FUNCTION_BLOCK FB_Example2

VAR
	fbRead1     :  FB_ReadAdsSymByName;
	bEnable     : BOOL;
	sSymbol     : STRING := 'GVL_Config.arrRack[1]';
	stStorageSlot : ST_StorageSlot;
	eComMode    :  E_AdsComMode := eAdsComModeFastCom;
	bBusy       : BOOL;
    bError      : BOOL;
    nErrId      : UDINT;
	bExecute: BOOL;
	fbTimer : TON := (PT := T#100MS); // Adjust the speed here
END_VAR


fbTimer(IN := NOT fbTimer.Q); // This creates a self-resetting pulse

IF fbTimer.Q THEN
    bEnable := TRUE; // Trigger your FB_ReadAdsSymByName
END_IF

	fbRead1(
	bRead:= bEnable, 
	sNetId:= '', 
	nPort:= 852, 
	sVarName:= sSymbol, 
	nDestAddr:= ADR(stStorageSlot), 
	nLen:= SIZEOF(stStorageSlot), 
	tTimeout:= , 
	eComMode:= eComMode,
	bBusy=> bBusy, 
	bError=> bError, 
	nErrorId=> nErrId);
bEnable := FALSE;

END_FUNCTION_BLOCK

(* stored: Version 1.1.0.1, ProductVersion 3.1.4024.16
   POU FB_Example2: Id {2261581c-2141-4e25-835b-2805700ea6a4}, SpecialFunc None *)
